# EPICS StreamDevice protocol: proto/scanivalveDts4050.proto
Terminator = "\r\n";

getString {
    in "\$1 %#s";
}

listVars {
    out "LIST \$1";
}

getIntVar {
    in "SET \$1 %d";
}

setIntVar {
    out "SET \$1 %d";
}

startScan {
    out "SET FORMAT 0";
    out "SET TIME 1";
    out "SCAN";
}

getScanFrameNum {
    in "Frame # %d";
}

getScanFrameTimeStamp {
    in "Time %d us";
}

getScanRtdTemp {
    ExtraInput = Ignore;
    in "Rtd\$1 %f %*s";
}

getScanUnits {
    in "Units %s";
}

getScanChTemp {
    in "\$1 %f %*s";
}

getScanChStatus {
    in "\$1 %*f %s";
}

sendCommand {
    out "\$1";
}
